ABB RobotStudio station: AssemblyCell_ZZRobotics_final.rspag

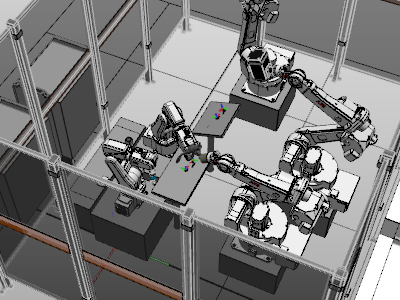
--- station ---
Station Project1 (saved by RobotStudio 22.3.10190.2)
Controller Controller4, task T_ROB2: task frame (RAPID world) sits at (-1070, 1330, 300) mm, rotated rx 0 ry 0 rz -90 deg in the station
Controller Controller4, task T_ROB1: task frame (RAPID world) sits at (-1070, 1330, 300) mm, rotated rx 0 ry 0 rz -90 deg in the station
Controller Controller3, task T_ROB1: task frame (RAPID world) sits at (-374.93, 1144.99, 305) mm, rotated rx 0 ry 0 rz -90 deg in the station
Controller Controller1, task T_ROB2: task frame (RAPID world) sits at (-250, 60, 415.69) mm, rotated rx 0 ry 0 rz 180 deg in the station
Controller Controller1, task T_ROB1: task frame (RAPID world) sits at (-250, 60, 415.69) mm, rotated rx 0 ry 0 rz 180 deg in the station
Controller Controller1
  mechanical unit ROB_1: IRB120_3_58__01_ActLoader, 6 joints, base frame (0, 0, 0) mm
  mechanical unit ROB_2: IRB120_3_58__01_ActTransmitter, 6 joints, base frame (588.39, -10, 0) mm, rotated rx 0 ry 0 rz -90 deg
Controller Controller3
  mechanical unit ROB_1: IRB1520ID_4_150__02_ActWelding, 6 joints, base frame (0, 0, 0) mm
Controller Controller4
  mechanical unit ROB_1: IRB1520ID_4_150__ActDrilling, 6 joints, base frame (0, 0, 0) mm
  mechanical unit ROB_2: IRB1520ID_4_150__ActEndeep, 6 joints, base frame (790, -930, 0) mm, rotated rx 0 ry 0 rz 90 deg
Layout (positions relative to the parent item):
  - RobotBase_Welding [part] at (-620, 914, 10) mm, size 500 x 500 x 300 mm
  - IRB120_3_58__01_ActTransmitter [mechanism, from Robots\IRB120_3_58_G_01.rslib] at (-838.39, 70, 415.69) mm, rotated rx 0 ry 0 rz 90 deg; joint values [-0.5895, 0.4014, 0.0311, 0, 1.1382, -2.1603] (rad or m)
  - IRB120_3_58__01_ActLoader [mechanism, from Robots\IRB120_3_58_G_01.rslib] at (-250, 60, 415.69) mm, rotated rx 0 ry 0 rz 180 deg; joint values [-1.4842, -0.4691, 0.5158, -0.0707, 1.4263, -0.6336] (rad or m)
  - Gripper_Vacuum [mechanism, from Components\smc_gripper.rslib] at (-261.42, 249.64, 930.86) mm, rotated rx -173.43 ry 2.1 rz -48.23 deg
  - Gripper_Fingers [mechanism, from Tools\ABB_Smart_Gripper_Servo_Fingers.rslib] at (-611, 410, 819.18) mm, rotated rx -180 ry 0 rz 0 deg; joint values [0] (rad or m)
  - RA_MTG4000_22 [mechanism, from Tools\Fronius_Robacta_MTG4000_22deg.rslib] at (-374.93, 698.3, 1167.59) mm, rotated rx 180 ry 55 rz 90 deg
  - Table_Welding [graphiccomponentgroup, from Components\Table_Welding.rslib] at (-730, 250, 0) mm
    - TableLeg [part, from Components\Table_Welding.rslib] at (110, 0, 0) mm
    - TablePlate [part, from Components\Table_Welding.rslib] at (730, -250, 0) mm
    - Cylinder_GripWelding_Support [mechanism, from Components\Cylinder.rslib] at (730, -250, 0) mm; joint values [0] (rad or m)
    - Cylinder_GripWelding_Tail [mechanism, from Components\Cylinder.rslib] at (-449, 580, 0) mm, rotated rx 0 ry 0 rz 180 deg; joint values [0] (rad or m)
  - Group_Inlet [graphiccomponentgroup] at (0, 3, 0) mm
    - Desk_L1_H1 [part] at (-279.56, -346.1, 404.98) mm, rotated rx 0 ry 0 rz 90 deg, size 60 x 90 x 5 mm
    - Desk_L2_H2 [part], size 100 x 60 x 5 mm
    - Profile_H1 [part] at (-683.6, -256.15, 395.47) mm, size 45 x 45 x 60 mm
    - Profile_H2 [part], size 45 x 45 x 70 mm
    - Table_Inlet [part] at (0, 40, 0) mm, size 1000 x 257.3 x 400 mm
    - l2_h2_welded [part] at (-595, 407, 640) mm, rotated rx 90 ry 0 rz 90 deg, size 60 x 75 x 100 mm
    - l1_h1_welded [part] at (-590, 407, 640) mm, rotated rx 0 ry 0 rz 90 deg, size 60 x 90 x 65 mm
    - l1_h1_welded_countersink [part] at (-1230, 404.46, 634.13) mm, rotated rx 90 ry -20 rz 90 deg, size 60 x 65 x 90 mm
    - l2_h2_welded_countersink [part] at (-1225, 404.46, 634.13) mm, rotated rx 90 ry -20 rz 90 deg, size 60 x 75 x 100 mm
    - l2_h2_welded_holes [part] at (-1225, 404.46, 634.13) mm, rotated rx 90 ry -20 rz 90 deg, size 60 x 75 x 100 mm
    - l1_h1_welded_holes [part] at (-1230, 404.46, 634.13) mm, rotated rx 90 ry -20 rz 90 deg, size 60 x 65 x 90 mm
    - Desk_L2_H2_1 [part], size 100 x 60 x 5 mm
    - Profile_H2_2 [part], size 45 x 45 x 70 mm
    - Desk_L2_H2_3 [part], size 100 x 60 x 5 mm
    - Profile_H2_4 [part], size 45 x 45 x 70 mm
    - Desk_L2_H2_5 [part], size 100 x 60 x 5 mm
    - Profile_H2_6 [part], size 45 x 45 x 70 mm
  - RobotBase_Transmission [part], size 500 x 500 x 404 mm
  - RobotBase_Loader [part] at (570, 0, 0) mm, size 500 x 500 x 404 mm
  - IRB1520ID_4_150__02_ActWelding [mechanism, from Robots\IRB1520ID_4_150_G_02.rslib] at (-374.93, 1144.99, 305) mm, rotated rx 0 ry 0 rz -90 deg; joint values [0, -1.2217, 1.0472, 0, 0.7854, 0] (rad or m)
  - SmartComponent_ActLoader [smart component]
      signals: DI do_grip_on, DI do_grip_off, DI do_vacuum_on, DI do_vacuum_off
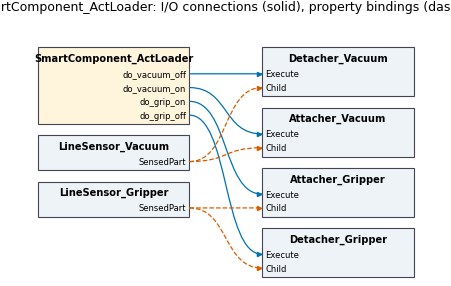
      connections:
        SmartComponent_ActLoader.do_vacuum_off -> Detacher_Vacuum.Execute
        SmartComponent_ActLoader.do_vacuum_on -> Attacher_Vacuum.Execute
        SmartComponent_ActLoader.do_grip_on -> Attacher_Gripper.Execute
        SmartComponent_ActLoader.do_grip_off -> Detacher_Gripper.Execute
        LineSensor_Vacuum.SensedPart => Detacher_Vacuum.Child
        LineSensor_Vacuum.SensedPart => Attacher_Vacuum.Child
        LineSensor_Gripper.SensedPart => Attacher_Gripper.Child
        LineSensor_Gripper.SensedPart => Detacher_Gripper.Child
    - LineSensor_Gripper [smart component, from Components\LineSensor.rslib] at (-611, 410, 704.98) mm, rotated rx -180 ry 0 rz 0 deg
        properties: Start=[0.000368147116492024 0.000112762068043337 -0.00954004890841353]; End=[0.000704727202270661 0.000672266486728079 0.0254538601137482]; Radius=0.005; SensedPart=(none); SensedPoint=[0 0 0]
      - _sensorPart_ [part], size 10.3 x 10.6 x 35.2 mm
    - LineSensor_Vacuum [smart component, from Components\LineSensor.rslib] at (-249.37, 270, 735.28) mm, rotated rx -173.43 ry 2.1 rz -48.23 deg
        properties: Start=[0.000258350395641593 -0.000244336751510213 0.000305598823163056]; End=[0.000624252122424396 0.000899619015264114 0.0102332108789397]; Radius=0.005; SensedPart=(none); SensedPoint=[-0.273905639648438 -0.353316131591797 0.454631866455078]
      - _sensorPart_ [part], size 10.1 x 10.9 x 11.1 mm
    - Attacher_Gripper [smart component, from Components\Attacher.rslib]
        properties: Parent=Gripper_Fingers; Flange=0; Child=(none); Mount=false; Offset=[0 0 0]; Orientation=[0 0 0]
    - Attacher_Vacuum [smart component, from Components\Attacher.rslib]
        properties: Parent=Gripper_Vacuum; Flange=0; Child=(none); Mount=false; Offset=[0 0 0]; Orientation=[0 0 0]
    - Detacher_Gripper [smart component, from Components\Detacher.rslib]
        properties: Child=(none); KeepPosition=true
    - Detacher_Vacuum [smart component, from Components\Detacher.rslib]
        properties: Child=(none); KeepPosition=true
  - SmartComponent_PartsIO [smart component]
      signals: DI spawn_desk_l1_h1, DI spawn_desk_l2_h2, DI spawn_profile_l1_h1, DI spawn_profile_l2_h2, DI spawn_welded_l1_h1, DI spawn_welded_l2_h2, DI spawn_holed_l1_h1, DI spawn_holed_l2_h2, DI drain_desk_l1_h1, DI drain_desk_l2_h2, DI drain_profile_l1_h1, DI drain_profile_l2_h2, DI drain_welded_l1_h1, DI drain_welded_l2_h2, DI drain_holed_l1_h1, DI drain_holed_l2_h2, DI drain_endeep_l2_h2, DI drain_endeep_l1_h1, DI spawn_endeep_l1_h1, DI spawn_endeep_l2_h2
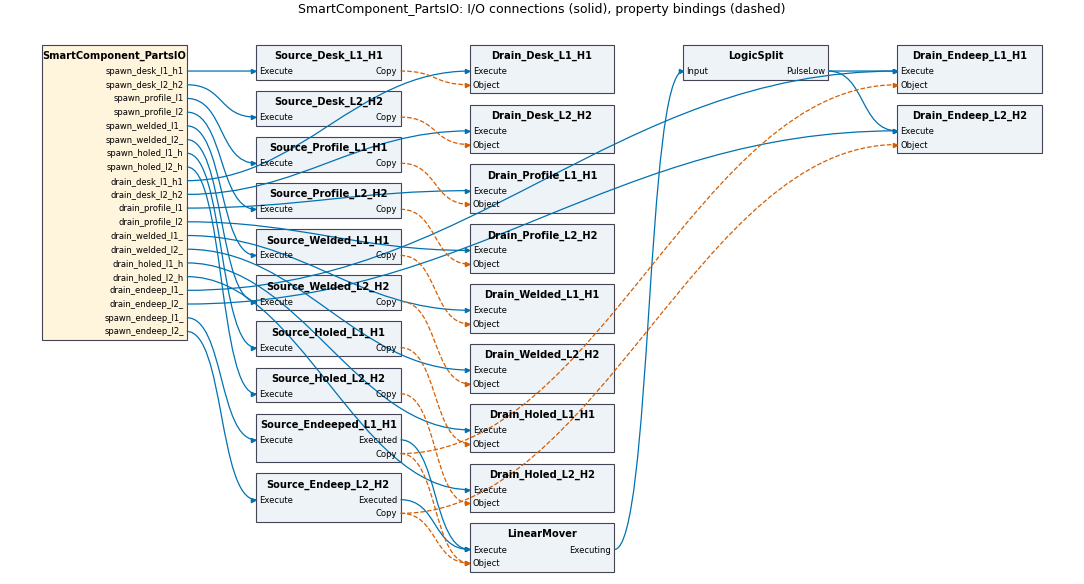
      connections:
        SmartComponent_PartsIO.spawn_desk_l1_h1 -> Source_Desk_L1_H1.Execute
        SmartComponent_PartsIO.spawn_desk_l2_h2 -> Source_Desk_L2_H2.Execute
        SmartComponent_PartsIO.spawn_profile_l1_h1 -> Source_Profile_L1_H1.Execute
        SmartComponent_PartsIO.spawn_profile_l2_h2 -> Source_Profile_L2_H2.Execute
        SmartComponent_PartsIO.spawn_welded_l1_h1 -> Source_Welded_L1_H1.Execute
        SmartComponent_PartsIO.spawn_welded_l2_h2 -> Source_Welded_L2_H2.Execute
        SmartComponent_PartsIO.spawn_holed_l1_h1 -> Source_Holed_L1_H1.Execute
        SmartComponent_PartsIO.spawn_holed_l2_h2 -> Source_Holed_L2_H2.Execute
        SmartComponent_PartsIO.drain_desk_l1_h1 -> Drain_Desk_L1_H1.Execute
        SmartComponent_PartsIO.drain_desk_l2_h2 -> Drain_Desk_L2_H2.Execute
        SmartComponent_PartsIO.drain_profile_l1_h1 -> Drain_Profile_L1_H1.Execute
        SmartComponent_PartsIO.drain_profile_l2_h2 -> Drain_Profile_L2_H2.Execute
        SmartComponent_PartsIO.drain_welded_l1_h1 -> Drain_Welded_L1_H1.Execute
        SmartComponent_PartsIO.drain_welded_l2_h2 -> Drain_Welded_L2_H2.Execute
        SmartComponent_PartsIO.drain_holed_l1_h1 -> Drain_Holed_L1_H1.Execute
        SmartComponent_PartsIO.drain_holed_l2_h2 -> Drain_Holed_L2_H2.Execute
        SmartComponent_PartsIO.drain_endeep_l1_h1 -> Drain_Endeep_L1_H1.Execute
        SmartComponent_PartsIO.drain_endeep_l2_h2 -> Drain_Endeep_L2_H2.Execute
        SmartComponent_PartsIO.spawn_endeep_l1_h1 -> Source_Endeeped_L1_H1.Execute
        SmartComponent_PartsIO.spawn_endeep_l2_h2 -> Source_Endeep_L2_H2.Execute
        Source_Endeep_L2_H2.Executed -> LinearMover.Execute
        Source_Endeeped_L1_H1.Executed -> LinearMover.Execute
        LinearMover.Executing -> LogicSplit.Input
        LogicSplit.PulseLow -> Drain_Endeep_L1_H1.Execute
        LogicSplit.PulseLow -> Drain_Endeep_L2_H2.Execute
        Source_Desk_L1_H1.Copy => Drain_Desk_L1_H1.Object
        Source_Desk_L2_H2.Copy => Drain_Desk_L2_H2.Object
        Source_Profile_L1_H1.Copy => Drain_Profile_L1_H1.Object
        Source_Profile_L2_H2.Copy => Drain_Profile_L2_H2.Object
        Source_Welded_L1_H1.Copy => Drain_Welded_L1_H1.Object
        Source_Welded_L2_H2.Copy => Drain_Welded_L2_H2.Object
        Source_Holed_L1_H1.Copy => Drain_Holed_L1_H1.Object
        Source_Holed_L2_H2.Copy => Drain_Holed_L2_H2.Object
        Source_Endeeped_L1_H1.Copy => Drain_Endeep_L1_H1.Object
        Source_Endeep_L2_H2.Copy => Drain_Endeep_L2_H2.Object
        Source_Endeeped_L1_H1.Copy => LinearMover.Object
        Source_Endeep_L2_H2.Copy => LinearMover.Object
    - Source_Desk_L1_H1 [smart component, from Components\Source.rslib] at (-294.16, -347, 399.98) mm, rotated rx 0 ry 0 rz 90 deg
        properties: Source=Desk_L1_H1; Copy=(none); Parent=(none); Position=[-0.279564 -0.346 0.404979]; Orientation=[0 0 1.5707963267949]; Transient=true; PhysicsBehavior=-1
    - Source_Desk_L2_H2 [smart component, from Components\Source.rslib]
        properties: Source=Desk_L2_H2; Copy=(none); Parent=(none); Position=[0 0 0]; Orientation=[0 0 0]; Transient=true; PhysicsBehavior=-1
    - Source_Profile_L1_H1 [smart component, from Components\Source.rslib]
        properties: Source=Profile_H1; Copy=(none); Parent=(none); Position=[-0.683597 -0.256153 0.395473]; Orientation=[0 0 0]; Transient=true; PhysicsBehavior=-1
    - Source_Profile_L2_H2 [smart component, from Components\Source.rslib]
        properties: Source=Profile_H2; Copy=(none); Parent=(none); Position=[0 0 0]; Orientation=[0 0 0]; Transient=true; PhysicsBehavior=-1
    - Source_Welded_L1_H1 [smart component, from Components\Source.rslib]
        properties: Source=l1_h1_welded; Copy=(none); Parent=(none); Position=[-0.59 0.407 0.64]; Orientation=[0 0 1.5707963267949]; Transient=true; PhysicsBehavior=-1
    - Source_Welded_L2_H2 [smart component, from Components\Source.rslib]
        properties: Source=l2_h2_welded; Copy=(none); Parent=(none); Position=[-0.595 0.407 0.64]; Orientation=[1.5707963267949 0 1.5707963267949]; Transient=true; PhysicsBehavior=-1
    - Source_Holed_L1_H1 [smart component, from Components\Source.rslib]
        properties: Source=l1_h1_welded_holes; Copy=(none); Parent=(none); Position=[-1.23 0.404459 0.634127]; Orientation=[1.5707963267949 -0.349065850398866 1.5707963267949]; Transient=true; PhysicsBehavior=-1
    - Source_Holed_L2_H2 [smart component, from Components\Source.rslib]
        properties: Source=l2_h2_welded_holes; Copy=(none); Parent=(none); Position=[-1.225 0.404459 0.634127]; Orientation=[1.5707963267949 -0.349065850398866 1.5707963267949]; Transient=true; PhysicsBehavior=-1
    - Drain_Desk_L1_H1 [smart component, from Components\Sink.rslib]
        properties: Object=(none)
    - Drain_Holed_L1_H1 [smart component, from Components\Sink.rslib]
        properties: Object=(none)
    - Drain_Profile_L2_H2 [smart component, from Components\Sink.rslib]
        properties: Object=(none)
    - Drain_Profile_L1_H1 [smart component, from Components\Sink.rslib]
        properties: Object=(none)
    - Drain_Welded_L2_H2 [smart component, from Components\Sink.rslib]
        properties: Object=(none)
    - Drain_Desk_L2_H2 [smart component, from Components\Sink.rslib]
        properties: Object=(none)
    - Drain_Holed_L2_H2 [smart component, from Components\Sink.rslib]
        properties: Object=(none)
    - Drain_Welded_L1_H1 [smart component, from Components\Sink.rslib]
        properties: Object=(none)
    - Source_Endeeped_L1_H1 [smart component, from Components\Source.rslib]
        properties: Source=l1_h1_welded_countersink; Copy=(none); Parent=(none); Position=[-1.23 0.404459 0.634127]; Orientation=[1.5707963267949 -0.349065850398866 1.5707963267949]; Transient=true; PhysicsBehavior=-1
    - Source_Endeep_L2_H2 [smart component, from Components\Source.rslib]
        properties: Source=l2_h2_welded_countersink; Copy=(none); Parent=(none); Position=[-1.225 0.404459 0.634127]; Orientation=[1.5707963267949 -0.349065850398866 1.5707963267949]; Transient=true; PhysicsBehavior=-1
    - Drain_Endeep_L2_H2 [smart component, from Components\Sink.rslib]
        properties: Object=(none)
    - Drain_Endeep_L1_H1 [smart component, from Components\Sink.rslib]
        properties: Object=(none)
    - LinearMover [smart component, from Components\LinearMover2.rslib]
        properties: Object=(none); Direction=[-0.1 0 0]; Distance=0.17; Duration=2; Reference=Local; ReferenceObject=(none)
    - LogicSplit [smart component, from Components\LogicSplit.rslib]
  - LogicGate [smart component, from Components\LogicGate.rslib]
      properties: Operator=AND; Delay=0
  - LogicGate_2 [smart component, from Components\LogicGate.rslib]
      properties: Operator=AND; Delay=0
  - LogicGate_3 [smart component, from Components\LogicGate.rslib]
      properties: Operator=AND; Delay=0
  - LogicGate_4 [smart component, from Components\LogicGate.rslib]
      properties: Operator=AND; Delay=0
  - Group_Drill_Endeep_Cell [graphiccomponentgroup]
    - RobotBase_Endeep [part] at (-1760, 283.99, 10) mm, rotated rx 0 ry 0 rz 90 deg, size 500 x 500 x 300 mm
    - RobotBase_Drilling [part] at (-1320, 1114, 10) mm, size 500 x 500 x 300 mm
    - Table_Drilling [graphiccomponentgroup] at (-1370, 250, 0) mm, rotated rx 20 ry 0 rz 0 deg
      - TableLeg [part] at (60, 0, 0) mm, rotated rx -20 ry 0 rz 0 deg, size 60 x 60 x 600 mm
      - TablePlate [part, from Components\TablePlate.rslib] at (1240, -234.92, 85.51) mm, rotated rx -20 ry 0 rz 0 deg
    - Cylinder_GripDrilling_Support [mechanism, from Components\Cylinder_1.rslib] at (-640, 240.97, -107.21) mm, rotated rx 20 ry 0 rz 0 deg; joint values [0] (rad or m)
    - Cylinder_GripDrilling_Tail [mechanism, from Components\Cylinder_1.rslib] at (-1819.91, 1021, 176.44) mm, rotated rx -20 ry 0 rz 180 deg; joint values [0] (rad or m)
    - Drill_Tool [mechanism, from Components\Drill_Tool.rslib] at (-1079.95, 911.09, 1539.96) mm, rotated rx -180 ry -70 rz -90 deg
    - Endeep_Tool [mechanism, from Components\Endeep_Tool.rslib] at (-1432.49, 333.31, 1851.39) mm, rotated rx 0 ry -70 rz -90 deg
  - IRB1520ID_4_150__ActDrilling [mechanism, from Robots\IRB1520ID_4_150_G_02.rslib] at (-1070, 1330, 300) mm, rotated rx 0 ry 0 rz -90 deg; joint values [-0.0458, -0.9578, 0.4598, 0.0574, 0.8482, -0.0537] (rad or m)
  - IRB1520ID_4_150__ActEndeep [mechanism, from Robots\IRB1520ID_4_150_G_02.rslib] at (-2000, 540, 300) mm; joint values [-0.6243, -0.1174, -0.2377, 2.1619, 1.978, -0.9764] (rad or m)
  - LogicGate_5 [smart component, from Components\LogicGate.rslib]
      properties: Operator=AND; Delay=0
  - LogicGate_6 [smart component, from Components\LogicGate.rslib]
      properties: Operator=AND; Delay=0
  - LogicGate_7 [smart component, from Components\LogicGate.rslib]
      properties: Operator=AND; Delay=0
  - LogicGate_8 [smart component, from Components\LogicGate.rslib]
      properties: Operator=AND; Delay=0
  - SmartComponent_Cylinders [smart component]
      signals: DI open_weld_support, DI open_weld_tail, DI open_drill_support, DI open_drill_tail, DI close_weld_support, DI close_weld_tail, DI close_drill_support, DI close_drill_tail
      connections:
        SmartComponent_Cylinders.open_drill_support -> PoseMover.Execute
        SmartComponent_Cylinders.close_drill_support -> PoseMover_2.Execute
        SmartComponent_Cylinders.open_drill_tail -> PoseMover_7.Execute
        SmartComponent_Cylinders.close_drill_tail -> PoseMover_3.Execute
        SmartComponent_Cylinders.open_weld_support -> PoseMover_6.Execute
        SmartComponent_Cylinders.close_weld_support -> PoseMover_4.Execute
        SmartComponent_Cylinders.open_weld_tail -> PoseMover_5.Execute
        SmartComponent_Cylinders.close_weld_tail -> PoseMover_8.Execute
    - PoseMover [smart component, from Components\PoseMover.rslib]
        properties: Mechanism=Cylinder_GripDrilling_Support; Pose=1; Duration=0
    - PoseMover_2 [smart component, from Components\PoseMover.rslib]
        properties: Mechanism=Cylinder_GripDrilling_Support; Pose=2; Duration=0
    - PoseMover_3 [smart component, from Components\PoseMover.rslib]
        properties: Mechanism=Cylinder_GripDrilling_Tail; Pose=2; Duration=0
    - PoseMover_4 [smart component, from Components\PoseMover.rslib]
        properties: Mechanism=Cylinder_GripWelding_Support; Pose=2; Duration=0
    - PoseMover_5 [smart component, from Components\PoseMover.rslib]
        properties: Mechanism=Cylinder_GripWelding_Tail; Pose=1; Duration=0
    - PoseMover_6 [smart component, from Components\PoseMover.rslib]
        properties: Mechanism=Cylinder_GripWelding_Support; Pose=1; Duration=0
    - PoseMover_7 [smart component, from Components\PoseMover.rslib]
        properties: Mechanism=Cylinder_GripDrilling_Tail; Pose=1; Duration=0
    - PoseMover_8 [smart component, from Components\PoseMover.rslib]
        properties: Mechanism=Cylinder_GripWelding_Tail; Pose=2; Duration=0
  - Fence [graphiccomponentgroup] at (0, 201.34, 0) mm
    - Z_Fence_800 [part] at (-2692.2, -847.39, 0) mm, size 159.8 x 979.2 x 2218.8 mm
    - Z_Fence_802 [part] at (-2692.2, 12.61, 0) mm, size 159.8 x 979.2 x 2218.8 mm
    - Z_Fence_806 [part] at (-2692.2, 872.87, 0) mm, size 159.8 x 979.2 x 2218.8 mm
    - Z_Fence_808 [part] at (-974.44, -853.03, 0) mm, rotated rx 0 ry 0 rz 90 deg, size 159.8 x 979.2 x 2218.8 mm
    - Z_Fence_809 [part] at (-1834.6, -853.03, 0) mm, rotated rx 0 ry 0 rz 90 deg, size 159.8 x 979.2 x 2218.8 mm
    - Z_Fence_810 [part] at (-114.19, -853.03, 0) mm, rotated rx 0 ry 0 rz 90 deg, size 159.8 x 979.2 x 2218.8 mm
    - Z_Fence_811 [part] at (745.69, -853.03, 0) mm, rotated rx 0 ry 0 rz 90 deg, size 159.8 x 979.2 x 2218.8 mm
    - Z_Fence_813 [part] at (-2691.02, 1743.1, 0) mm, rotated rx 0 ry 0 rz -90 deg, size 159.8 x 979.2 x 2218.8 mm
    - Z_Fence_814 [part] at (-1830.85, 1743.1, 0) mm, rotated rx 0 ry 0 rz -90 deg, size 159.8 x 979.2 x 2218.8 mm
    - Z_Fence_815 [part] at (-110.06, 1743.1, 0) mm, rotated rx 0 ry 0 rz -90 deg, size 159.8 x 979.2 x 2218.8 mm
    - Z_Fence_816 [part] at (-970.7, 1743.1, 0) mm, rotated rx 0 ry 0 rz -90 deg, size 159.8 x 979.2 x 2218.8 mm
    - Z_Fence_818 [part] at (749.49, 1737.83, 0) mm, rotated rx 0 ry 0 rz 180 deg, size 159.8 x 979.2 x 2218.8 mm
    - Z_Fence_819 [part] at (749.49, 877.62, 0) mm, rotated rx 0 ry 0 rz 180 deg, size 159.8 x 979.2 x 2218.8 mm
    - Z_Fence_820 [part] at (749.49, 17.63, 0) mm, rotated rx 0 ry 0 rz 180 deg, size 159.8 x 979.2 x 2218.8 mm
  - _Skrine [graphiccomponentgroup]
    - OmniCore V250XT [mechanism, from %ABB.RobotStudio.Models.OmniCore%\OmniCore_V250XT.rslib] at (-135.27, 2273.01, 0) mm, rotated rx 0 ry 0 rz 180 deg; joint values [0] (rad or m)
    - OmniCore V250XT_2 [mechanism, from %ABB.RobotStudio.Models.OmniCore%\OmniCore_V250XT.rslib] at (-930.19, 2273.01, 0) mm, rotated rx 0 ry 0 rz 180 deg; joint values [0] (rad or m)
    - OmniCore V250XT_3 [mechanism, from %ABB.RobotStudio.Models.OmniCore%\OmniCore_V250XT.rslib] at (-1769.47, 2273.01, 0) mm, rotated rx 0 ry 0 rz 180 deg; joint values [0] (rad or m)
    - OmniCore V250XT_4 [mechanism, from %ABB.RobotStudio.Models.OmniCore%\OmniCore_V250XT.rslib] at (-51.9, -1005.58, 0) mm; joint values [0] (rad or m)
    - OmniCore V250XT_5 [mechanism, from %ABB.RobotStudio.Models.OmniCore%\OmniCore_V250XT.rslib] at (-880.12, -1005.58, 0) mm; joint values [0] (rad or m)
Attachment: Gripper_Vacuum is attached to IRB120_3_58__01_ActLoader / Link6
Attachment: Gripper_Fingers is attached to IRB120_3_58__01_ActTransmitter / Link6
Attachment: RA_MTG4000_22 is attached to IRB1520ID_4_150__02_ActWelding / Link6
Attachment: LineSensor_Gripper is attached to Gripper_Fingers / HandBase
Attachment: LineSensor_Vacuum is attached to Gripper_Vacuum / Assembly_ABBGRIP_2
Attachment: Drill_Tool is attached to IRB1520ID_4_150__ActDrilling / Link6
Attachment: Endeep_Tool is attached to IRB1520ID_4_150__ActEndeep / Link6
Station signals: DI p_type_1_small, DI p_type_2_big, DI produce
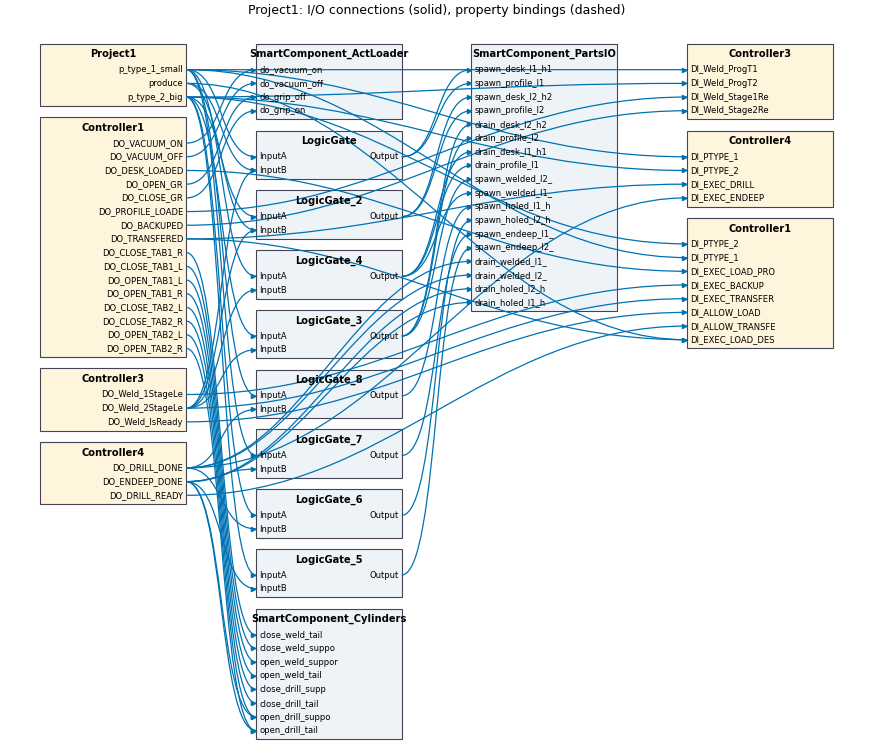
Station logic (signal -> signal, property => property):
  Project1.p_type_1_small -> LogicGate.InputA
  Project1.produce -> LogicGate.InputB
  LogicGate.Output -> SmartComponent_PartsIO.spawn_desk_l1_h1
  LogicGate.Output -> SmartComponent_PartsIO.spawn_profile_l1_h1
  Project1.p_type_2_big -> LogicGate_2.InputA
  Project1.produce -> LogicGate_2.InputB
  LogicGate_2.Output -> SmartComponent_PartsIO.spawn_desk_l2_h2
  LogicGate_2.Output -> SmartComponent_PartsIO.spawn_profile_l2_h2
  Controller1.DO_VACUUM_ON -> SmartComponent_ActLoader.do_vacuum_on
  Controller1.DO_VACUUM_OFF -> SmartComponent_ActLoader.do_vacuum_off
  Project1.p_type_2_big -> Controller1.DI_PTYPE_2
  Project1.p_type_1_small -> Controller1.DI_PTYPE_1
  Controller1.DO_DESK_LOADED -> Controller1.DI_EXEC_LOAD_PROFILE
  Controller1.DO_OPEN_GR -> SmartComponent_ActLoader.do_grip_off
  Controller1.DO_CLOSE_GR -> SmartComponent_ActLoader.do_grip_on
  Project1.p_type_1_small -> Controller3.DI_Weld_ProgT1
  Project1.p_type_2_big -> Controller3.DI_Weld_ProgT2
  Controller1.DO_PROFILE_LOADED -> Controller3.DI_Weld_Stage1Req
  Controller3.DO_Weld_1StageLeave -> Controller1.DI_EXEC_BACKUP
  Controller1.DO_BACKUPED -> Controller3.DI_Weld_Stage2Req
  Controller3.DO_Weld_2StageLeave -> Controller1.DI_EXEC_TRANSFER
  Project1.p_type_2_big -> LogicGate_3.InputA
  Controller3.DO_Weld_2StageLeave -> LogicGate_3.InputB
  LogicGate_3.Output -> SmartComponent_PartsIO.drain_desk_l2_h2
  LogicGate_3.Output -> SmartComponent_PartsIO.drain_profile_l2_h2
  Project1.p_type_1_small -> LogicGate_4.InputA
  Controller3.DO_Weld_2StageLeave -> LogicGate_4.InputB
  LogicGate_4.Output -> SmartComponent_PartsIO.drain_desk_l1_h1
  LogicGate_4.Output -> SmartComponent_PartsIO.drain_profile_l1_h1
  LogicGate_3.Output -> SmartComponent_PartsIO.spawn_welded_l2_h2
  LogicGate_4.Output -> SmartComponent_PartsIO.spawn_welded_l1_h1
  Project1.p_type_1_small -> Controller4.DI_PTYPE_1
  Project1.p_type_2_big -> Controller4.DI_PTYPE_2
  Controller1.DO_TRANSFERED -> Controller4.DI_EXEC_DRILL
  Controller4.DO_DRILL_DONE -> Controller4.DI_EXEC_ENDEEP
  Project1.p_type_1_small -> LogicGate_8.InputA
  Project1.p_type_2_big -> LogicGate_6.InputA
  Controller4.DO_DRILL_DONE -> LogicGate_8.InputB
  Controller4.DO_DRILL_DONE -> LogicGate_6.InputB
  Project1.p_type_1_small -> LogicGate_7.InputA
  Project1.p_type_2_big -> LogicGate_5.InputA
  Controller4.DO_ENDEEP_DONE -> LogicGate_7.InputB
  Controller4.DO_ENDEEP_DONE -> LogicGate_5.InputB
  LogicGate_8.Output -> SmartComponent_PartsIO.spawn_holed_l1_h1
  LogicGate_6.Output -> SmartComponent_PartsIO.spawn_holed_l2_h2
  LogicGate_7.Output -> SmartComponent_PartsIO.spawn_endeep_l1_h1
  LogicGate_5.Output -> SmartComponent_PartsIO.spawn_endeep_l2_h2
  Controller1.DO_CLOSE_TAB1_R -> SmartComponent_Cylinders.close_weld_tail
  Controller1.DO_CLOSE_TAB1_L -> SmartComponent_Cylinders.close_weld_support
  Controller1.DO_OPEN_TAB1_L -> SmartComponent_Cylinders.open_weld_support
  Controller1.DO_OPEN_TAB1_R -> SmartComponent_Cylinders.open_weld_tail
  Controller1.DO_CLOSE_TAB2_L -> SmartComponent_Cylinders.close_drill_support
  Controller1.DO_CLOSE_TAB2_R -> SmartComponent_Cylinders.close_drill_tail
  Controller1.DO_OPEN_TAB2_L -> SmartComponent_Cylinders.open_drill_support
  Controller1.DO_OPEN_TAB2_R -> SmartComponent_Cylinders.open_drill_tail
  Controller4.DO_ENDEEP_DONE -> SmartComponent_Cylinders.open_drill_tail
  Controller4.DO_ENDEEP_DONE -> SmartComponent_Cylinders.open_drill_support
  Controller3.DO_Weld_IsReady -> Controller1.DI_ALLOW_LOAD
  Controller3.DO_Weld_2StageLeave -> LogicGate_2.InputB
  Controller3.DO_Weld_2StageLeave -> LogicGate.InputB
  Controller4.DO_DRILL_READY -> Controller1.DI_ALLOW_TRANSFER
  Project1.produce -> Controller1.DI_EXEC_LOAD_DESK
  Controller1.DO_TRANSFERED -> Controller1.DI_EXEC_LOAD_DESK
  Controller4.DO_DRILL_DONE -> SmartComponent_PartsIO.drain_welded_l1_h1
  Controller4.DO_DRILL_DONE -> SmartComponent_PartsIO.drain_welded_l2_h2
  Controller4.DO_ENDEEP_DONE -> SmartComponent_PartsIO.drain_holed_l2_h2
  Controller4.DO_ENDEEP_DONE -> SmartComponent_PartsIO.drain_holed_l1_h1
Targets, tools, work objects and paths stored in the station and not in the controller backup, written as RAPID:
! task T_ROB2
MODULE Module1
  CONST num WaitGripper:=1;
ENDMODULE


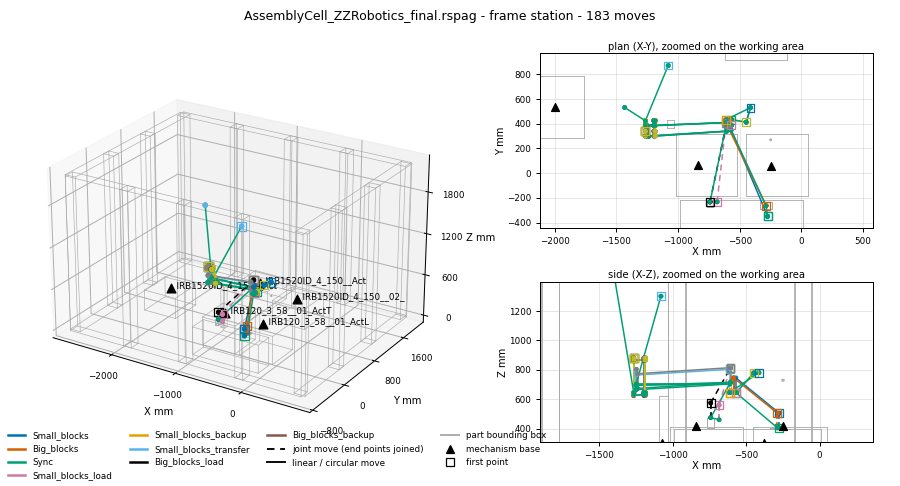
[picture p0: tool path of AssemblyCell_ZZRobotics_final.rspag in frame station, 183 of 212 moves have a stored position in this frame; points joined in program order, loops and branches not executed]
--- Controller Data/Controller1/RAPID/TASK1/PROGMOD/CalibData.mod ---
MODULE CalibData
    PERS tooldata Gripper_Vacuum:=[TRUE,[[0,0.004,197.001],[1,0,0,0]],[1,[0.207,-0.496,71.18],[1,0,0,0],0,0,0]];
ENDMODULE

--- Controller Data/Controller1/RAPID/TASK1/PROGMOD/Module1.mod ---
MODULE Module1
    CONST jointtarget Target_JHome:=[[-85.037200714,-26.876673148,29.555461388,-4.048831126,81.721717608,-36.301936344],[9E+09,9E+09,9E+09,9E+09,9E+09,9E+09]];

    CONST robtarget Target_Base_l2_h2:=[[36.607,323.865,-10.716],[0,0,1,0],[0,0,0,0],[9E+09,9E+09,9E+09,9E+09,9E+09,9E+09]];
    CONST robtarget Target_Base_l1_h1:=[[24.164,410,-10.605],[0,0,1,0],[0,0,1,0],[9E+09,9E+09,9E+09,9E+09,9E+09,9E+09]];

    CONST robtarget Target_Table1_l2_h2_pre:=[[335,-293,229.805],[0,0,1,0],[-1,-1,0,0],[9E+09,9E+09,9E+09,9E+09,9E+09,9E+09]];
    CONST robtarget Target_Table1_l2_h2:=[[335,-346.85,229.340933033],[0,0,1,0],[-1,-1,0,0],[9E+09,9E+09,9E+09,9E+09,9E+09,9E+09]];

    CONST robtarget Target_Table1_l1_h1_pre:=[[319.886,-290.252,229.772],[0,0,1,0],[0,0,0,0],[9E+09,9E+09,9E+09,9E+09,9E+09,9E+09]];
    CONST robtarget Target_Table1_l1_h1:=[[334.586,-342.952,229.372],[0,0,1,0],[0,0,0,0],[9E+09,9E+09,9E+09,9E+09,9E+09,9E+09]];

    VAR bool cold_start:=TRUE;
    CONST num wait_vacuum:=1;

    PROC main()
        IF cold_start THEN
            Init;
            cold_start:=FALSE;
        ENDIF

        WaitDI DI_EXEC_LOAD_DESK,1;
        WaitDI DI_ALLOW_LOAD,1;

        IF TestDI(DI_PTYPE_1) THEN
            Small_blocks;
        ELSEIF TestDI(DI_PTYPE_2) THEN
            Big_blocks;
        ELSE
            RETURN ;
        ENDIF
    ENDPROC

    PROC Init()
        PulseDO DO_OPEN_TAB1_L;
        PulseDO DO_OPEN_TAB1_R;
        MoveAbsJ Target_JHome,v1000,fine,Gripper_Vacuum\WObj:=wobj0;
    ENDPROC

    PROC Small_blocks()
        MoveJ Offs(Target_Base_l1_h1,0,0,100),v1000,fine,Gripper_Vacuum;
        MoveJ Offs(Target_Base_l1_h1,0,0,0),v1000,fine,Gripper_Vacuum;

        !Attach %%%%%%%%%%%%%%%%%%%%%%%%%%%%%%%%%%%%%%
        PulseDO DO_VACUUM_ON;
        WaitTime wait_vacuum;

        MoveJ Offs(Target_Base_l1_h1,0,0,100),v1000,fine,Gripper_Vacuum;
        MoveL Offs(Target_Table1_l1_h1_pre,0,0,100),v1000,fine,Gripper_Vacuum;
        WaitTime 0.5;
        MoveL Offs(Target_Table1_l1_h1_pre,0,0,0),v200,fine,Gripper_Vacuum;
        WaitTime 0.5;
        MoveL Offs(Target_Table1_l1_h1,0,0,0),v200,fine,Gripper_Vacuum;

        WaitTime 0.5;
        PulseDO DO_CLOSE_TAB1_L;
        PulseDO DO_CLOSE_TAB1_R;

        !Detach %%%%%%%%%%%%%%%%
        PulseDO DO_VACUUM_OFF;
        WaitTime wait_vacuum;

        MoveL Offs(Target_Table1_l1_h1,0,0,100),v200,fine,Gripper_Vacuum;
        MoveAbsJ Target_JHome,v1000,fine,Gripper_Vacuum\WObj:=wobj0;

        PulseDO DO_DESK_LOADED;
    ENDPROC

    PROC Big_blocks()
        MoveJ Offs(Target_Base_l2_h2,0,0,100),v1000,fine,Gripper_Vacuum;
        MoveJ Offs(Target_Base_l2_h2,0,0,0),v1000,fine,Gripper_Vacuum;

        !Attach %%%%%%%%%%%%%%%%%%%%%%%%%%%%%%%%%%%%%%
        PulseDO DO_VACUUM_ON;
        WaitTime wait_vacuum;

        MoveJ Offs(Target_Base_l2_h2,0,0,100),v1000,fine,Gripper_Vacuum;
        MoveL Offs(Target_Table1_l2_h2_pre,0,0,100),v1000,fine,Gripper_Vacuum;
        WaitTime 0.5;
        MoveL Offs(Target_Table1_l2_h2_pre,0,0,0),v200,fine,Gripper_Vacuum;
        WaitTime 0.5;
        MoveL Offs(Target_Table1_l2_h2,0,0,0),v200,fine,Gripper_Vacuum;

        WaitTime 0.5;
        PulseDO DO_CLOSE_TAB1_L;
        PulseDO DO_CLOSE_TAB1_R;

        !Detach %%%%%%%%%%%%%%%%
        PulseDO DO_VACUUM_OFF;
        WaitTime wait_vacuum;

        MoveL Offs(Target_Table1_l2_h2,0,0,100),v200,fine,Gripper_Vacuum;
        MoveAbsJ Target_JHome,v1000,fine,Gripper_Vacuum\WObj:=wobj0;

        PulseDO DO_DESK_LOADED;
    ENDPROC

    PROC Sync()
        MoveAbsJ Target_JHome,v1000,fine,Gripper_Vacuum\WObj:=wobj0;
        MoveL Target_Base_l1_h1,v1000,z100,Gripper_Vacuum\WObj:=wobj0;
        MoveL Target_Base_l2_h2,v1000,z100,Gripper_Vacuum\WObj:=wobj0;
        MoveL Target_Table1_l1_h1_pre,v1000,z100,Gripper_Vacuum\WObj:=wobj0;
        MoveL Target_Table1_l1_h1,v1000,z100,Gripper_Vacuum\WObj:=wobj0;
        MoveL Target_Table1_l2_h2_pre,v1000,z100,Gripper_Vacuum\WObj:=wobj0;
        MoveL Target_Table1_l2_h2,v1000,z100,Gripper_Vacuum\WObj:=wobj0;
    ENDPROC
ENDMODULE

--- Controller Data/Controller1/RAPID/TASK2/PROGMOD/CalibData.mod ---
MODULE CalibData
    PERS tooldata Gripper_Fingers:=[TRUE,[[0,0,114.2],[1,0,0,0]],[0.215,[8.7,12.3,49.2],[1,0,0,0],0.00021,0.00024,0.00009]];
ENDMODULE

--- Controller Data/Controller1/RAPID/TASK2/PROGMOD/Module1.mod ---
MODULE Module1
    CONST jointtarget Target_JHome:=[[-26.597577745,-44.264017247,35.261659694,-19.248693519,81.614947173,-88.381493558],[9E+09,9E+09,9E+09,9E+09,9E+09,9E+09]];

    CONST robtarget Target_Base_l2_h2:=[[490.966,292.847,59.284],[0,0.707106781,0.707106781,0],[-2,0,0,0],[9E+09,9E+09,9E+09,9E+09,9E+09,9E+09]];
    CONST robtarget Target_Base_l1_h1:=[[433.597,292.153,44.778],[0,0.707106781,0.707106781,0],[-2,0,1,0],[9E+09,9E+09,9E+09,9E+09,9E+09,9E+09]];

    CONST robtarget Target_Table1_l1_h1_takeout:=[[360.972830849,-280.009480233,288.1717752],[0.004810357,-0.000232941,0.999956482,-0.007990003],[-1,0,-2,0],[9E+09,9E+09,9E+09,9E+09,9E+09,9E+09]];
    CONST robtarget Target_Table1_l2_h2_takeout:=[[356,-280,299.305],[0,0,1,0],[-1,0,-2,0],[9E+09,9E+09,9E+09,9E+09,9E+09,9E+09]];

    CONST robtarget Target_Table1_l2_h2:=[[356,-350,299.305],[0,0,1,0],[-1,0,-2,0],[9E+09,9E+09,9E+09,9E+09,9E+09,9E+09]];
    CONST robtarget Target_Table1_l1_h1:=[[361,-350.001,289.29],[0,0,1,0],[-1,0,-2,0],[9E+09,9E+09,9E+09,9E+09,9E+09,9E+09]];

    CONST robtarget Target_Table2_l1_h1:=[[1001,-325.091129765,279.687062196],[0,0,0.984807753,-0.173648178],[0,-1,0,0],[9E+09,9E+09,9E+09,9E+09,9E+09,9E+09]];
    CONST robtarget Target_Table2_l2_h2:=[[996,-321.807256971,288.908661883],[0,0,0.984807753,-0.173648178],[0,0,0,0],[9E+09,9E+09,9E+09,9E+09,9E+09,9E+09]];

    CONST robtarget Target_Table2_l2_h2_takeout:=[[988.5,-237.234921117,258.126848932],[0,0,0.984807753,-0.173648178],[0,0,0,0],[9E+09,9E+09,9E+09,9E+09,9E+09,9E+09]];
    CONST robtarget Target_Table2_l1_h1_takeout:=[[999.5,-240.655323444,248.729567219],[0,0,0.984807753,-0.173648178],[0,-1,0,0],[9E+09,9E+09,9E+09,9E+09,9E+09,9E+09]];

    VAR bool cold_start:=TRUE;
    CONST num wait_gripper:=1;

    PROC main()
        IF cold_start THEN
            Init;
            cold_start:=FALSE;
        ENDIF

        WaitDI DI_EXEC_LOAD_PROFILE,1;
        WaitDI DI_ALLOW_LOAD,1;

        IF TestDI(DI_PTYPE_1) THEN
            Small_blocks_load;
            WaitDI DI_EXEC_BACKUP,1;
            Small_blocks_backup;
            WaitDI DI_EXEC_TRANSFER,1;
            WaitDI DI_ALLOW_TRANSFER,1;
            Small_blocks_transfer;
        ELSEIF TestDI(DI_PTYPE_2) THEN
            Big_blocks_load;
            WaitDI DI_EXEC_BACKUP,1;
            Big_blocks_backup;
            WaitDI DI_EXEC_TRANSFER,1;
            WaitDI DI_ALLOW_TRANSFER,1;
            Big_blocks_transfer;
        ELSE
            RETURN ;
        ENDIF
    ENDPROC

    PROC Init()
        PulseDO DO_OPEN_GR;
        PulseDO DO_OPEN_TAB2_L;
        PulseDO DO_OPEN_TAB2_R;

        MoveAbsJ Target_JHome,v1000,fine,Gripper_Fingers\WObj:=wobj0;
    ENDPROC

    PROC Small_blocks_load()
        MoveJ Offs(Target_Base_l1_h1,0,0,100),v1000,fine,Gripper_Fingers;

        !OPEN Gripper
        PulseDO DO_OPEN_GR;
        WaitTime wait_gripper;

        MoveJ Offs(Target_Base_l1_h1,0,0,0),v1000,fine,Gripper_Fingers;

        !Close gripper
        PulseDO DO_CLOSE_GR;
        WaitTime wait_gripper;

        MoveJ Offs(Target_Base_l1_h1,0,0,100),v1000,fine,Gripper_Fingers;
        MoveJ Offs(Target_Table1_l1_h1,0,0,100),v1000,fine,Gripper_Fingers;
        MoveJ Target_Table1_l1_h1,v200,fine,Gripper_Fingers;
        WaitTime 0.5;

        PulseDO DO_PROFILE_LOADED;
    ENDPROC

    PROC Small_blocks_backup()
        !OPEN Gripper
        PulseDO DO_OPEN_GR;
        WaitTime wait_gripper;

        MoveJ Offs(Target_Table1_l1_h1,0,0,100),v200,fine,Gripper_Fingers;
        MoveAbsJ Target_JHome,v1000,fine,Gripper_Fingers\WObj:=wobj0;

        PulseDO DO_BACKUPED;
    ENDPROC

    PROC Small_blocks_transfer()
        !OPEN Gripper
        PulseDO DO_OPEN_GR;
        WaitTime wait_gripper;

        MoveJ Offs(Target_Table1_l1_h1,0,0,100),v1000,fine,Gripper_Fingers;
        MoveJ Target_Table1_l1_h1,v200,fine,Gripper_Fingers;
        WaitTime 0.5;

        PulseDO DO_OPEN_TAB1_L;
        PulseDO DO_OPEN_TAB1_R;

        !Close gripper
        PulseDO DO_CLOSE_GR;
        WaitTime wait_gripper;

        MoveL Target_Table1_l1_h1_takeout,v200,fine,Gripper_Fingers;
        MoveL Offs(Target_Table1_l1_h1_takeout,0,0,100),v1000,fine,Gripper_Fingers;

        MoveL Offs(Target_Table2_l1_h1_takeout,0,0,100),v1000,fine,Gripper_Fingers;
        MoveL Offs(Target_Table2_l1_h1_takeout,0,0,0),v200,fine,Gripper_Fingers;
        MoveL Offs(Target_Table2_l1_h1,0,0,0),v200,fine,Gripper_Fingers;
        WaitTime 0.5;

        PulseDO DO_CLOSE_TAB2_L;
        PulseDO DO_CLOSE_TAB2_R;

        PulseDO DO_OPEN_GR;
        WaitTime wait_gripper;

        MoveL Offs(Target_Table2_l1_h1,0,0,100),v1000,fine,Gripper_Fingers;
        MoveAbsJ Target_JHome,v1000,fine,Gripper_Fingers\WObj:=wobj0;

        PulseDO DO_TRANSFERED;
    ENDPROC

    PROC Big_blocks_load()
        MoveJ Offs(Target_Base_l2_h2,0,0,100),v1000,fine,Gripper_Fingers;

        !OPEN Gripper
        PulseDO DO_OPEN_GR;
        WaitTime wait_gripper;

        MoveJ Offs(Target_Base_l2_h2,0,0,0),v1000,fine,Gripper_Fingers;
        !Close gripper
        PulseDO DO_CLOSE_GR;
        WaitTime wait_gripper;

        MoveJ Offs(Target_Base_l2_h2,0,0,100),v1000,fine,Gripper_Fingers;
        MoveJ Offs(Target_Table1_l2_h2,0,0,100),v1000,fine,Gripper_Fingers;
        MoveJ Offs(Target_Table1_l2_h2,0,0,0),v200,fine,Gripper_Fingers;

        PulseDO DO_PROFILE_LOADED;
    ENDPROC

    PROC Big_blocks_backup()
        !OPEN Gripper
        PulseDO DO_OPEN_GR;
        WaitTime wait_gripper;

        MoveJ Offs(Target_Table1_l2_h2,0,0,100),v200,fine,Gripper_Fingers;
        MoveAbsJ Target_JHome,v1000,fine,Gripper_Fingers\WObj:=wobj0;

        PulseDO DO_BACKUPED;
    ENDPROC

    PROC Big_blocks_transfer()
        !OPEN Gripper
        PulseDO DO_OPEN_GR;
        WaitTime wait_gripper;

        MoveJ Offs(Target_Table1_l2_h2,0,0,100),v1000,fine,Gripper_Fingers;
        MoveJ Target_Table1_l2_h2,v200,fine,Gripper_Fingers;
        WaitTime 0.5;

        PulseDO DO_OPEN_TAB1_L;
        PulseDO DO_OPEN_TAB1_R;

        !Close gripper
        PulseDO DO_CLOSE_GR;
        WaitTime wait_gripper;

        MoveL Target_Table1_l2_h2_takeout,v200,fine,Gripper_Fingers;
        MoveL Offs(Target_Table1_l2_h2_takeout,0,0,100),v1000,fine,Gripper_Fingers;

        MoveL Offs(Target_Table2_l2_h2_takeout,0,0,100),v1000,fine,Gripper_Fingers;
        MoveL Offs(Target_Table2_l2_h2_takeout,0,0,0),v200,fine,Gripper_Fingers;
        MoveL Offs(Target_Table2_l2_h2,0,0,0),v200,fine,Gripper_Fingers;

        !Detach
        PulseDO DO_CLOSE_TAB2_L;
        PulseDO DO_CLOSE_TAB2_R;

        PulseDO DO_OPEN_GR;
        WaitTime wait_gripper;

        MoveL Offs(Target_Table2_l2_h2,0,0,100),v1000,fine,Gripper_Fingers;
        MoveAbsJ Target_JHome,v1000,fine,Gripper_Fingers\WObj:=wobj0;

        PulseDO DO_TRANSFERED;
    ENDPROC
    PROC Sync()
        MoveAbsJ Target_JHome,v1000,fine,Gripper_Fingers\WObj:=wobj0;
        MoveL Target_Base_l1_h1,v1000,z100,Gripper_Fingers\WObj:=wobj0;
        MoveL Target_Base_l2_h2,v1000,z100,Gripper_Fingers\WObj:=wobj0;
        MoveL Target_Table1_l2_h2,v1000,z100,Gripper_Fingers\WObj:=wobj0;
        MoveL Target_Table2_l1_h1,v1000,z100,Gripper_Fingers\WObj:=wobj0;
        MoveL Target_Table1_l1_h1,v1000,z100,Gripper_Fingers\WObj:=wobj0;
        MoveL Target_Table2_l2_h2,v1000,z100,Gripper_Fingers\WObj:=wobj0;
        MoveL Target_Table2_l2_h2_takeout,v1000,z100,Gripper_Fingers\WObj:=wobj0;
        MoveL Target_Table1_l2_h2_takeout,v1000,z100,Gripper_Fingers\WObj:=wobj0;
        MoveL Target_Table1_l1_h1_takeout,v1000,z100,Gripper_Fingers\WObj:=wobj0;
        MoveL Target_Table2_l1_h1_takeout,v1000,z100,Gripper_Fingers\WObj:=wobj0;
    ENDPROC
ENDMODULE

--- Controller Data/Controller3/RAPID/TASK1/PROGMOD/CalibData.mod ---
MODULE CalibData
    PERS tooldata Weldgun:=[TRUE,[[20.31,0,363.689],[0.948464781,0,0.316882565,0]],[1,[0,0,1],[1,0,0,0],0,0,0]];
ENDMODULE

--- Controller Data/Controller3/RAPID/TASK1/PROGMOD/Module1.mod ---
MODULE Module1
    CONST jointtarget Target_Idle:=[[0,-70,60,0,45,0],[9E+09,9E+09,9E+09,9E+09,9E+09,9E+09]];

    CONST robtarget Target_20_2:=[[711.495384789,-192.569070764,340],[0.270598049,0.653281483,-0.653281483,0.27059805],[-1,-1,-2,0],[9E+09,9E+09,9E+09,9E+09,9E+09,9E+09]];
    CONST robtarget Target_30_2:=[[756.495384789,-192.569070764,340],[0.270598049,0.653281483,-0.653281483,0.27059805],[-1,-1,-2,0],[9E+09,9E+09,9E+09,9E+09,9E+09,9E+09]];
    CONST robtarget Target_30:=[[756.495384789,-192.569070764,340],[0.45999152,0.077308088,-0.883635489,0.040244043],[-1,-1,-1,0],[9E+09,9E+09,9E+09,9E+09,9E+09,9E+09]];
    CONST robtarget Target_40:=[[756.495384789,-237.569070764,340],[0.382683432,0,-0.923879533,0],[-1,-1,-1,0],[9E+09,9E+09,9E+09,9E+09,9E+09,9E+09]];
    CONST robtarget Target_40_2:=[[756.495384789,-237.569070764,340],[0.27059805,-0.653281483,-0.653281483,-0.27059805],[-1,0,0,0],[9E+09,9E+09,9E+09,9E+09,9E+09,9E+09]];
    CONST robtarget Target_10_2:=[[711.495384789,-237.569070764,340],[0.270598048,-0.653281483,-0.653281483,-0.27059805],[-1,0,0,0],[9E+09,9E+09,9E+09,9E+09,9E+09,9E+09]];
    CONST robtarget Target_10:=[[711.495384789,-237.569070764,340],[0.176703546,-0.819491154,-0.33944435,-0.426600093],[-1,0,1,0],[9E+09,9E+09,9E+09,9E+09,9E+09,9E+09]];
    CONST robtarget Target_20:=[[711.495384789,-192.569070764,340],[-0.000000001,0.923879533,0,0.382683432],[-1,0,1,0],[9E+09,9E+09,9E+09,9E+09,9E+09,9E+09]];
    CONST robtarget Target_10_30_0:=[[614.316010633,-38.379402252,476.187474664],[0.146446608,-0.853553391,-0.353553391,-0.353553391],[-1,0,1,0],[9E+09,9E+09,9E+09,9E+09,9E+09,9E+09]];
    CONST robtarget Target_10_30_1:=[[731.697116217,-72.603148817,474.139403279],[0.379409522,-0.049950211,-0.915975615,0.120590478],[-1,-1,-1,0],[9E+09,9E+09,9E+09,9E+09,9E+09,9E+09]];

    VAR speeddata welding := v150;
    CONST num PType1Offs:=0;
    CONST num PType2Offs:=5;

    VAR bool ColdStart:=TRUE;
    VAR num PTypeRequested;

    PROC main()
        IF ColdStart THEN
            SetDO DO_Weld_IsReady,0;
            SetDO DO_Weld_IsBusy,1;

            MoveAbsJ Target_Idle,v1000,fine,Weldgun\WObj:=wobj0;

            SetDO DO_Weld_IsReady,1;
            SetDO DO_Weld_IsBusy,0;
            ColdStart := FALSE;
        ENDIF

        WaitDI DI_Weld_Stage1Req,1;

        IF TestDI(DI_Weld_ProgT1) THEN
            PTypeRequested:=1;
        ELSEIF TestDI(DI_Weld_ProgT2) THEN
            PTypeRequested:=2;
        ENDIF

        SetDO DO_Weld_IsReady,0;
        SetDO DO_Weld_IsBusy,1;

        PulseDO DO_Weld_1StageEnter;
        Path_10_30 PTypeRequested;
        PulseDO DO_Weld_1StageLeave;

        WaitDI DI_Weld_Stage2Req,1;

        PulseDO DO_Weld_2StageEnter;
        Path_20_30_40_10 PTypeRequested;
        PulseDO DO_Weld_2StageLeave;

        SetDO DO_Weld_IsBusy,0;
        SetDO DO_Weld_IsReady,1;
    ENDPROC

    FUNC robtarget ResolvePtype(robtarget Target,num PType)
        TEST PType
        CASE 1:
            RETURN Offs(Target,0,PType1Offs,0);
        CASE 2:
            RETURN Offs(Target,0,PType2Offs,0);
        DEFAULT:
            RETURN Target;
        ENDTEST
    ENDFUNC

    PROC Path_20_30_40_10(num PType)
        MoveAbsJ Target_Idle,v1000,fine,Weldgun\WObj:=wobj0;

        MoveL Target_10_30_1,v1000,z50,Weldgun\WObj:=wobj0;
        MoveL Offs(Target_20_2,0,10,10),v1000,z100,Weldgun\WObj:=wobj0;

        WaitTime 1;
        MoveL ResolvePtype(Target_20_2,PType),welding,z100,Weldgun\WObj:=wobj0;
        MoveL ResolvePtype(Target_30_2,PType),welding,z100,Weldgun\WObj:=wobj0;
        WaitTime 1;

        MoveL ResolvePtype(Target_30,PType),welding,z100,Weldgun\WObj:=wobj0;
        MoveL ResolvePtype(Target_40,PType),welding,z100,Weldgun\WObj:=wobj0;
        WaitTime 1;
        MoveL ResolvePtype(Target_40_2,PType),welding,z100,Weldgun\WObj:=wobj0;
        MoveL ResolvePtype(Target_10_2,PType),welding,z100,Weldgun\WObj:=wobj0;
        WaitTime 1;
        MoveL ResolvePtype(Target_10,PType),welding,z100,Weldgun\WObj:=wobj0;
        MoveL ResolvePtype(Target_20,PType),welding,z100,Weldgun\WObj:=wobj0;

        MoveL Target_10_30_0,v1000,z50,Weldgun\WObj:=wobj0;

        MoveAbsJ Target_Idle,v1000,fine,Weldgun\WObj:=wobj0;
    ENDPROC

    PROC Path_10_30(num PType)
        MoveAbsJ Target_Idle,v1000,fine,Weldgun\WObj:=wobj0;

        MoveL Target_10_30_0,v1000,z10,Weldgun\WObj:=wobj0;

        MoveL ResolvePtype(Offs(Target_10,-10,0,10),PType),v800,fine,Weldgun\WObj:=wobj0;
        MoveL ResolvePtype(Target_10,PType),welding,fine,Weldgun\WObj:=wobj0;
        WaitTime 0.5;
        MoveL ResolvePtype(Offs(Target_10,-10,0,10),PType),welding,fine,Weldgun\WObj:=wobj0;

        MoveL Target_10_30_0,v1000,z10,Weldgun\WObj:=wobj0;
        MoveL Target_10_30_1,v1000,z10,Weldgun\WObj:=wobj0;

        MoveL ResolvePtype(Offs(Target_30,10,10,10),PType),v800,fine,Weldgun\WObj:=wobj0;
        MoveL ResolvePtype(Target_30,PType),welding,fine,Weldgun\WObj:=wobj0;
        WaitTime 0.5;
        MoveL ResolvePtype(Offs(Target_30,10,10,10),PType),welding,fine,Weldgun\WObj:=wobj0;

        MoveL Target_10_30_1,v1000,z10,Weldgun\WObj:=wobj0;
        MoveAbsJ Target_Idle,v1000,fine,Weldgun\WObj:=wobj0;
    ENDPROC

    PROC Path_10_20()
        MoveL Target_10,welding,fine,Weldgun\WObj:=wobj0;
        MoveL Target_20,welding,fine,Weldgun\WObj:=wobj0;
    ENDPROC

    PROC Path_20_30()
        MoveL Target_20_2,welding,fine,Weldgun\WObj:=wobj0;
        MoveL Target_30_2,welding,fine,Weldgun\WObj:=wobj0;
    ENDPROC

    PROC Path_30_40()
        MoveL Target_30,welding,fine,Weldgun\WObj:=wobj0;
        MoveL Target_40,welding,fine,Weldgun\WObj:=wobj0;
    ENDPROC

    PROC Path_40_10()
        MoveL Target_10_2,welding,fine,Weldgun\WObj:=wobj0;
        MoveL Target_40_2,welding,fine,Weldgun\WObj:=wobj0;
    ENDPROC
    PROC Sync()
        MoveL Target_10,v1000,z100,Weldgun\WObj:=wobj0;
        MoveL Target_10_2,v1000,z100,Weldgun\WObj:=wobj0;
        MoveL Target_10_30_0,v1000,z100,Weldgun\WObj:=wobj0;
        MoveL Target_10_30_1,v1000,z100,Weldgun\WObj:=wobj0;
        MoveL Target_20,v1000,z100,Weldgun\WObj:=wobj0;
        MoveL Target_20_2,v1000,z100,Weldgun\WObj:=wobj0;
        MoveL Target_30,v1000,z100,Weldgun\WObj:=wobj0;
        MoveL Target_30_2,v1000,z100,Weldgun\WObj:=wobj0;
        MoveL Target_40,v1000,z100,Weldgun\WObj:=wobj0;
        MoveL Target_40_2,v1000,z100,Weldgun\WObj:=wobj0;
    ENDPROC
ENDMODULE

--- Controller Data/Controller4/RAPID/TASK1/PROGMOD/CalibData.mod ---
MODULE CalibData
    PERS tooldata Drill_Tool:=[TRUE,[[211.187000005,0.000000004,132.999999995],[0.707106781,0,0.707106781,0]],[1,[-40.884000001,0.010000002,112.464],[1,0,0,0],0,0,0]];
ENDMODULE

--- Controller Data/Controller4/RAPID/TASK1/PROGMOD/Module1.mod ---
MODULE Module1
    CONST robtarget T_Drill_aHome:=[[457.561710524,-9.948272227,1001.147802577],[0.173648178,0,-0.984807753,0],[0,0,0,0],[9E+09,9E+09,9E+09,9E+09,9E+09,9E+09]];
    CONST robtarget T_Drill_COM_10:=[[905.457950428,-195,345.666062685],[0.160429997,-0.376869611,-0.909843726,0.066452281],[0,-1,1,0],[9E+09,9E+09,9E+09,9E+09,9E+09,9E+09]];
    CONST robtarget T_Drill_COM_20:=[[943.045950428,-195,331.985062685],[0.160429997,-0.376869611,-0.909843726,0.066452281],[0,-1,1,0],[9E+09,9E+09,9E+09,9E+09,9E+09,9E+09]];
    CONST robtarget T_Drill_S_30:=[[943.045950428,-125,331.985062685],[0.160429997,-0.376869611,-0.909843726,0.066452281],[0,-1,1,0],[9E+09,9E+09,9E+09,9E+09,9E+09,9E+09]];
    CONST robtarget T_Drill_S_40:=[[905.457950428,-125,345.666062685],[0.160429997,-0.376869611,-0.909843726,0.066452281],[0,-1,1,0],[9E+09,9E+09,9E+09,9E+09,9E+09,9E+09]];
    CONST robtarget T_Drill_L_30:=[[943.045950428,-115,331.985062685],[0.160429997,-0.376869611,-0.909843726,0.066452281],[0,-1,1,0],[9E+09,9E+09,9E+09,9E+09,9E+09,9E+09]];
    CONST robtarget T_Drill_L_40:=[[905.457950428,-115,345.666062685],[0.160429997,-0.376869611,-0.909843726,0.066452281],[0,-1,1,0],[9E+09,9E+09,9E+09,9E+09,9E+09,9E+09]];

    VAR speeddata vel_move := v800;
    VAR speeddata vel_drill := v50;
    VAR speeddata vel_gotohole := v500;
    VAR num offset := -250;
    VAR num drillhole := 7;

    VAR bool COLD_START:=TRUE;

    PROC main()
        IF COLD_START THEN
            MoveL RelTool(T_Drill_aHome, 0, 0, 0),vel_move,fine,Drill_Tool\WObj:=wobj0;
            COLD_START := FALSE;
            SetDO DO_DRILL_READY,1;
        ENDIF

        WaitDI DI_EXEC_DRILL,1;
        SetDO DO_DRILL_READY,0;

        IF TestDI(DI_PTYPE_1) THEN
            Path_Drill_S;
            MoveL RelTool(T_Drill_aHome, 0, 0, 0),vel_move,fine,Drill_Tool\WObj:=wobj0;
            PulseDO DO_DRILL_DONE;
        ELSEIF TestDI(DI_PTYPE_2) THEN
            Path_Drill_L;
            MoveL RelTool(T_Drill_aHome, 0, 0, 0),vel_move,fine,Drill_Tool\WObj:=wobj0;
            PulseDO DO_DRILL_DONE;
        ELSE
            RETURN ;
        ENDIF
    ENDPROC

    PROC Path_Drill_S()
        MoveL RelTool(T_Drill_COM_10, 0, 0, offset),vel_move,fine,Drill_Tool\WObj:=wobj0;
        MoveL RelTool(T_Drill_COM_10, 0, 0, 0),vel_gotohole,fine,Drill_Tool\WObj:=wobj0;
        WaitTime 0.5;
        MoveL RelTool(T_Drill_COM_10, 0, 0, drillhole),vel_drill,fine,Drill_Tool\WObj:=wobj0;
        MoveL RelTool(T_Drill_COM_10, 0, 0, 0),vel_drill,fine,Drill_Tool\WObj:=wobj0;
        WaitTime 0.5;
        MoveL RelTool(T_Drill_COM_10, 0, 0, offset),vel_gotohole,fine,Drill_Tool\WObj:=wobj0;

        MoveL RelTool(T_Drill_COM_20, 0, 0, offset),vel_move,fine,Drill_Tool\WObj:=wobj0;
        MoveL RelTool(T_Drill_COM_20, 0, 0, 0),vel_gotohole,fine,Drill_Tool\WObj:=wobj0;
        WaitTime 0.5;
        MoveL RelTool(T_Drill_COM_20, 0, 0, drillhole),vel_drill,fine,Drill_Tool\WObj:=wobj0;
        MoveL RelTool(T_Drill_COM_20, 0, 0, 0),vel_drill,fine,Drill_Tool\WObj:=wobj0;
        WaitTime 0.5;
        MoveL RelTool(T_Drill_COM_20, 0, 0, offset),vel_gotohole,fine,Drill_Tool\WObj:=wobj0;

        MoveL RelTool(T_Drill_S_30, 0, 0, offset),vel_move,fine,Drill_Tool\WObj:=wobj0;
        MoveL RelTool(T_Drill_S_30, 0, 0, 0),vel_gotohole,fine,Drill_Tool\WObj:=wobj0;
        WaitTime 0.5;
        MoveL RelTool(T_Drill_S_30, 0, 0, drillhole),vel_drill,fine,Drill_Tool\WObj:=wobj0;
        MoveL RelTool(T_Drill_S_30, 0, 0, 0),vel_drill,fine,Drill_Tool\WObj:=wobj0;
        WaitTime 0.5;
        MoveL RelTool(T_Drill_S_30, 0, 0, offset),vel_gotohole,fine,Drill_Tool\WObj:=wobj0;

        MoveL RelTool(T_Drill_S_40, 0, 0, offset),vel_move,fine,Drill_Tool\WObj:=wobj0;
        MoveL RelTool(T_Drill_S_40, 0, 0, 0),vel_gotohole,fine,Drill_Tool\WObj:=wobj0;
        WaitTime 0.5;
        MoveL RelTool(T_Drill_S_40, 0, 0, drillhole),vel_drill,fine,Drill_Tool\WObj:=wobj0;
        MoveL RelTool(T_Drill_S_40, 0, 0, 0),vel_drill,fine,Drill_Tool\WObj:=wobj0;
        WaitTime 0.5;
        MoveL RelTool(T_Drill_S_40, 0, 0, offset),vel_gotohole,fine,Drill_Tool\WObj:=wobj0;

        !MoveL T_Drill_aHome,v200,fine,Drill_Tool\WObj:=wobj0;
        !MoveL T_Drill_COM_10,v200,fine,Drill_Tool\WObj:=wobj0;
        !MoveL T_Drill_COM_20,v200,fine,Drill_Tool\WObj:=wobj0;
        !MoveL T_Drill_S_30,v200,fine,Drill_Tool\WObj:=wobj0;
        !MoveL T_Drill_S_40,v200,fine,Drill_Tool\WObj:=wobj0;
    ENDPROC

    PROC Path_Drill_L()
        MoveL RelTool(T_Drill_COM_10, 0, 0, offset),vel_move,fine,Drill_Tool\WObj:=wobj0;
        MoveL RelTool(T_Drill_COM_10, 0, 0, 0),vel_gotohole,fine,Drill_Tool\WObj:=wobj0;
        WaitTime 0.5;
        MoveL RelTool(T_Drill_COM_10, 0, 0, drillhole),vel_drill,fine,Drill_Tool\WObj:=wobj0;
        MoveL RelTool(T_Drill_COM_10, 0, 0, 0),vel_drill,fine,Drill_Tool\WObj:=wobj0;
        WaitTime 0.5;
        MoveL RelTool(T_Drill_COM_10, 0, 0, offset),vel_gotohole,fine,Drill_Tool\WObj:=wobj0;

        MoveL RelTool(T_Drill_COM_20, 0, 0, offset),vel_move,fine,Drill_Tool\WObj:=wobj0;
        MoveL RelTool(T_Drill_COM_20, 0, 0, 0),vel_gotohole,fine,Drill_Tool\WObj:=wobj0;
        WaitTime 0.5;
        MoveL RelTool(T_Drill_COM_20, 0, 0, drillhole),vel_drill,fine,Drill_Tool\WObj:=wobj0;
        MoveL RelTool(T_Drill_COM_20, 0, 0, 0),vel_drill,fine,Drill_Tool\WObj:=wobj0;
        WaitTime 0.5;
        MoveL RelTool(T_Drill_COM_20, 0, 0, offset),vel_gotohole,fine,Drill_Tool\WObj:=wobj0;

        MoveL RelTool(T_Drill_L_30, 0, 0, offset),vel_move,fine,Drill_Tool\WObj:=wobj0;
        MoveL RelTool(T_Drill_L_30, 0, 0, 0),vel_gotohole,fine,Drill_Tool\WObj:=wobj0;
        WaitTime 0.5;
        MoveL RelTool(T_Drill_L_30, 0, 0, drillhole),vel_drill,fine,Drill_Tool\WObj:=wobj0;
        MoveL RelTool(T_Drill_L_30, 0, 0, 0),vel_drill,fine,Drill_Tool\WObj:=wobj0;
        WaitTime 0.5;
        MoveL RelTool(T_Drill_L_30, 0, 0, offset),vel_gotohole,fine,Drill_Tool\WObj:=wobj0;

        MoveL RelTool(T_Drill_L_40, 0, 0, offset),vel_move,fine,Drill_Tool\WObj:=wobj0;
        MoveL RelTool(T_Drill_L_40, 0, 0, 0),vel_gotohole,fine,Drill_Tool\WObj:=wobj0;
        WaitTime 0.5;
        MoveL RelTool(T_Drill_L_40, 0, 0, drillhole),vel_drill,fine,Drill_Tool\WObj:=wobj0;
        MoveL RelTool(T_Drill_L_40, 0, 0, 0),vel_drill,fine,Drill_Tool\WObj:=wobj0;
        WaitTime 0.5;
        MoveL RelTool(T_Drill_L_40, 0, 0, offset),vel_gotohole,fine,Drill_Tool\WObj:=wobj0;

        !MoveL T_Drill_aHome,v200,fine,Drill_Tool\WObj:=wobj0;
        !MoveL T_Drill_COM_10,v200,fine,Drill_Tool\WObj:=wobj0;
        !MoveL T_Drill_COM_20,v200,fine,Drill_Tool\WObj:=wobj0;
        !MoveL T_Drill_L_30,v200,fine,Drill_Tool\WObj:=wobj0;
        !MoveL T_Drill_L_40,v200,fine,Drill_Tool\WObj:=wobj0;
    ENDPROC

    PROC Sync()
        MoveL T_Drill_aHome,v200,fine,Drill_Tool\WObj:=wobj0;
        MoveL T_Drill_COM_10,v200,fine,Drill_Tool\WObj:=wobj0;
        MoveL T_Drill_COM_20,v200,fine,Drill_Tool\WObj:=wobj0;
        MoveL T_Drill_S_30,v200,fine,Drill_Tool\WObj:=wobj0;
        MoveL T_Drill_S_40,v200,fine,Drill_Tool\WObj:=wobj0;
        MoveL T_Drill_L_30,v200,fine,Drill_Tool\WObj:=wobj0;
        MoveL T_Drill_L_40,v200,fine,Drill_Tool\WObj:=wobj0;
    ENDPROC

ENDMODULE

--- Controller Data/Controller4/RAPID/TASK2/PROGMOD/CalibData.mod ---
MODULE CalibData
    PERS tooldata Endeep_Tool:=[TRUE,[[257.929,0,133],[0.707106781,0,0.707106781,0]],[1,[40.263,-0.01,112.48],[1,0,0,0],0,0,0]];
ENDMODULE

--- Controller Data/Controller4/RAPID/TASK2/PROGMOD/Module1.mod ---
MODULE Module1
    CONST robtarget T_Endeep_aHome:=[[797.552204235,-362.673625766,1349.391204212],[0,0.984807753,0,-0.173648178],[0,0,0,0],[9E+09,9E+09,9E+09,9E+09,9E+09,9E+09]];
    CONST robtarget T_Endeep_COM_10:=[[905.458,-195,345.666],[0,0.984807753,0,-0.173648178],[-1,0,-2,0],[9E+09,9E+09,9E+09,9E+09,9E+09,9E+09]];
    CONST robtarget T_Endeep_COM_20:=[[943.046,-195,331.985],[0,0.984807753,0,-0.173648178],[-1,0,-2,0],[9E+09,9E+09,9E+09,9E+09,9E+09,9E+09]];
    CONST robtarget T_Endeep_S_30:=[[943.046,-125,331.985],[0,0.984807753,0,-0.173648178],[-1,0,-2,0],[9E+09,9E+09,9E+09,9E+09,9E+09,9E+09]];
    CONST robtarget T_Endeep_S_40:=[[905.458,-125,345.666],[0,0.984807753,0,-0.173648178],[-1,0,-2,0],[9E+09,9E+09,9E+09,9E+09,9E+09,9E+09]];
    CONST robtarget T_Endeep_L_30:=[[943.046,-115,331.985],[0,0.984807753,0,-0.173648178],[-1,0,-2,0],[9E+09,9E+09,9E+09,9E+09,9E+09,9E+09]];
    CONST robtarget T_Endeep_L_40:=[[905.458,-115,345.666],[0,0.984807753,0,-0.173648178],[-1,0,-2,0],[9E+09,9E+09,9E+09,9E+09,9E+09,9E+09]];

    VAR speeddata vel_move:=v800;
    VAR speeddata vel_drill:=v50;
    VAR speeddata vel_gotohole:=v500;
    VAR num offset:=-250;
    VAR num endeephole:=2.5;

    VAR bool COLD_START:=TRUE;

    PROC main()
        IF COLD_START THEN
            MoveL RelTool(T_Endeep_aHome, 0, 0, 0),vel_move,fine,Endeep_Tool\WObj:=wobj0;
            COLD_START := FALSE;
        ENDIF

        WaitDI DI_EXEC_ENDEEP,1;

        IF TestDI(DI_PTYPE_1) THEN
            Path_Endeep_S;
            MoveL RelTool(T_Endeep_aHome, 0, 0, 0),vel_move,fine,Endeep_Tool\WObj:=wobj0;
            PulseDO DO_ENDEEP_DONE;
        ELSEIF TestDI(DI_PTYPE_2) THEN
            Path_Endeep_L;
            MoveL RelTool(T_Endeep_aHome, 0, 0, 0),vel_move,fine,Endeep_Tool\WObj:=wobj0;
            PulseDO DO_ENDEEP_DONE;
        ELSE
            RETURN ;
        ENDIF

        PulseDO DO_ENDEEP_DONE;
        SetDO DO_DRILL_READY,1;

    ENDPROC

    PROC Path_Endeep_S()
        MoveL RelTool(T_Endeep_COM_10,0,0,offset),vel_move,fine,Endeep_Tool\WObj:=wobj0;
        MoveL RelTool(T_Endeep_COM_10,0,0,0),vel_gotohole,fine,Endeep_Tool\WObj:=wobj0;
        WaitTime 0.5;
        MoveL RelTool(T_Endeep_COM_10,0,0,endeephole),vel_drill,fine,Endeep_Tool\WObj:=wobj0;
        MoveL RelTool(T_Endeep_COM_10,0,0,0),vel_drill,fine,Endeep_Tool\WObj:=wobj0;
        WaitTime 0.5;
        MoveL RelTool(T_Endeep_COM_10,0,0,offset),vel_gotohole,fine,Endeep_Tool\WObj:=wobj0;

        MoveL RelTool(T_Endeep_COM_20,0,0,offset),vel_move,fine,Endeep_Tool\WObj:=wobj0;
        MoveL RelTool(T_Endeep_COM_20,0,0,0),vel_gotohole,fine,Endeep_Tool\WObj:=wobj0;
        WaitTime 0.5;
        MoveL RelTool(T_Endeep_COM_20,0,0,endeephole),vel_drill,fine,Endeep_Tool\WObj:=wobj0;
        MoveL RelTool(T_Endeep_COM_20,0,0,0),vel_drill,fine,Endeep_Tool\WObj:=wobj0;
        WaitTime 0.5;
        MoveL RelTool(T_Endeep_COM_20,0,0,offset),vel_gotohole,fine,Endeep_Tool\WObj:=wobj0;

        MoveL RelTool(T_Endeep_S_30,0,0,offset),vel_move,fine,Endeep_Tool\WObj:=wobj0;
        MoveL RelTool(T_Endeep_S_30,0,0,0),vel_gotohole,fine,Endeep_Tool\WObj:=wobj0;
        WaitTime 0.5;
        MoveL RelTool(T_Endeep_S_30,0,0,endeephole),vel_drill,fine,Endeep_Tool\WObj:=wobj0;
        MoveL RelTool(T_Endeep_S_30,0,0,0),vel_drill,fine,Endeep_Tool\WObj:=wobj0;
        WaitTime 0.5;
        MoveL RelTool(T_Endeep_S_30,0,0,offset),vel_gotohole,fine,Endeep_Tool\WObj:=wobj0;

        MoveL RelTool(T_Endeep_S_40,0,0,offset),vel_move,fine,Endeep_Tool\WObj:=wobj0;
        MoveL RelTool(T_Endeep_S_40,0,0,0),vel_gotohole,fine,Endeep_Tool\WObj:=wobj0;
        WaitTime 0.5;
        MoveL RelTool(T_Endeep_S_40,0,0,endeephole),vel_drill,fine,Endeep_Tool\WObj:=wobj0;
        MoveL RelTool(T_Endeep_S_40,0,0,0),vel_drill,fine,Endeep_Tool\WObj:=wobj0;
        WaitTime 0.5;
        MoveL RelTool(T_Endeep_S_40,0,0,offset),vel_gotohole,fine,Endeep_Tool\WObj:=wobj0;

        !MoveL T_Endeep_aHome,v200,fine,Endeep_Tool\WObj:=wobj0;
        !MoveL T_Endeep_COM_10,v200,fine,Endeep_Tool\WObj:=wobj0;
        !MoveL T_Endeep_COM_20,v200,fine,Endeep_Tool\WObj:=wobj0;
        !MoveL T_Endeep_S_30,v200,fine,Endeep_Tool\WObj:=wobj0;
        !MoveL T_Endeep_S_40,v200,fine,Endeep_Tool\WObj:=wobj0;
    ENDPROC

    PROC Path_Endeep_L()
        MoveL RelTool(T_Endeep_COM_10,0,0,offset),vel_move,fine,Endeep_Tool\WObj:=wobj0;
        MoveL RelTool(T_Endeep_COM_10,0,0,0),vel_gotohole,fine,Endeep_Tool\WObj:=wobj0;
        WaitTime 0.5;
        MoveL RelTool(T_Endeep_COM_10,0,0,endeephole),vel_drill,fine,Endeep_Tool\WObj:=wobj0;
        MoveL RelTool(T_Endeep_COM_10,0,0,0),vel_drill,fine,Endeep_Tool\WObj:=wobj0;
        WaitTime 0.5;
        MoveL RelTool(T_Endeep_COM_10,0,0,offset),vel_gotohole,fine,Endeep_Tool\WObj:=wobj0;

        MoveL RelTool(T_Endeep_COM_20,0,0,offset),vel_move,fine,Endeep_Tool\WObj:=wobj0;
        MoveL RelTool(T_Endeep_COM_20,0,0,0),vel_gotohole,fine,Endeep_Tool\WObj:=wobj0;
        WaitTime 0.5;
        MoveL RelTool(T_Endeep_COM_20,0,0,endeephole),vel_drill,fine,Endeep_Tool\WObj:=wobj0;
        MoveL RelTool(T_Endeep_COM_20,0,0,0),vel_drill,fine,Endeep_Tool\WObj:=wobj0;
        WaitTime 0.5;
        MoveL RelTool(T_Endeep_COM_20,0,0,offset),vel_gotohole,fine,Endeep_Tool\WObj:=wobj0;

        MoveL RelTool(T_Endeep_L_30,0,0,offset),vel_move,fine,Endeep_Tool\WObj:=wobj0;
        MoveL RelTool(T_Endeep_L_30,0,0,0),vel_gotohole,fine,Endeep_Tool\WObj:=wobj0;
        WaitTime 0.5;
        MoveL RelTool(T_Endeep_L_30,0,0,endeephole),vel_drill,fine,Endeep_Tool\WObj:=wobj0;
        MoveL RelTool(T_Endeep_L_30,0,0,0),vel_drill,fine,Endeep_Tool\WObj:=wobj0;
        WaitTime 0.5;
        MoveL RelTool(T_Endeep_L_30,0,0,offset),vel_gotohole,fine,Endeep_Tool\WObj:=wobj0;

        MoveL RelTool(T_Endeep_L_40,0,0,offset),vel_move,fine,Endeep_Tool\WObj:=wobj0;
        MoveL RelTool(T_Endeep_L_40,0,0,0),vel_gotohole,fine,Endeep_Tool\WObj:=wobj0;
        WaitTime 0.5;
        MoveL RelTool(T_Endeep_L_40,0,0,endeephole),vel_drill,fine,Endeep_Tool\WObj:=wobj0;
        MoveL RelTool(T_Endeep_L_40,0,0,0),vel_drill,fine,Endeep_Tool\WObj:=wobj0;
        WaitTime 0.5;
        MoveL RelTool(T_Endeep_L_40,0,0,offset),vel_gotohole,fine,Endeep_Tool\WObj:=wobj0;

        !MoveL T_Endeep_aHome,v200,fine,Endeep_Tool\WObj:=wobj0;
        !MoveL T_Endeep_COM_10,v200,fine,Endeep_Tool\WObj:=wobj0;
        !MoveL T_Endeep_COM_20,v200,fine,Endeep_Tool\WObj:=wobj0;
        !MoveL T_Endeep_L_30,v200,fine,Endeep_Tool\WObj:=wobj0;
        !MoveL T_Endeep_L_40,v200,fine,Endeep_Tool\WObj:=wobj0;
    ENDPROC

    PROC Sync()
        MoveL T_Endeep_aHome,v200,fine,Endeep_Tool\WObj:=wobj0;
        MoveL T_Endeep_COM_10,v200,fine,Endeep_Tool\WObj:=wobj0;
        MoveL T_Endeep_COM_20,v200,fine,Endeep_Tool\WObj:=wobj0;
        MoveL T_Endeep_S_30,v200,fine,Endeep_Tool\WObj:=wobj0;
        MoveL T_Endeep_S_40,v200,fine,Endeep_Tool\WObj:=wobj0;
        MoveL T_Endeep_L_30,v200,fine,Endeep_Tool\WObj:=wobj0;
        MoveL T_Endeep_L_40,v200,fine,Endeep_Tool\WObj:=wobj0;
    ENDPROC
ENDMODULE

--- Controller Data/Controller1/SYSPAR/EIO.cfg ---
EIO:CFG_1.0:6:1::
#
EIO_SIGNAL:

      -Name "DO_OPEN_TAB1_L" -SignalType "DO"

      -Name "DO_OPEN_TAB1_R" -SignalType "DO"

      -Name "DO_CLOSE_TAB1_L" -SignalType "DO"

      -Name "DO_CLOSE_TAB1_R" -SignalType "DO"

      -Name "DO_CLOSE_TAB2_L" -SignalType "DO"

      -Name "DO_CLOSE_TAB2_R" -SignalType "DO"

      -Name "DO_OPEN_TAB2_L" -SignalType "DO"

      -Name "DO_OPEN_TAB2_R" -SignalType "DO"

      -Name "DO_OPEN_GR" -SignalType "DO"

      -Name "DO_CLOSE_GR" -SignalType "DO"

      -Name "DI_PTYPE_2" -SignalType "DI"

      -Name "DI_PTYPE_1" -SignalType "DI"

      -Name "DI_EXEC_LOAD_DESK" -SignalType "DI"

      -Name "DI_EXEC_LOAD_PROFILE" -SignalType "DI"

      -Name "DI_EXEC_TRANSFER" -SignalType "DI"

      -Name "DO_VACUUM_ON" -SignalType "DO"

      -Name "DO_VACUUM_OFF" -SignalType "DO"

      -Name "DO_DESK_LOADED" -SignalType "DO"

      -Name "DO_PROFILE_LOADED" -SignalType "DO"

      -Name "DI_EXEC_BACKUP" -SignalType "DI"

      -Name "DO_BACKUPED" -SignalType "DO"

      -Name "DO_TRANSFERED" -SignalType "DO"

      -Name "DI_ALLOW_LOAD" -SignalType "DI"

      -Name "DI_ALLOW_TRANSFER" -SignalType "DI"

--- Controller Data/Controller3/SYSPAR/EIO.cfg ---
EIO:CFG_1.0:6:1::
#
EIO_SIGNAL:

      -Name "DO_Weld_IsReady" -SignalType "DO"

      -Name "DO_Weld_IsBusy" -SignalType "DO"

      -Name "DO_Weld_1StageWip" -SignalType "DO"

      -Name "DO_Weld_2StageWip" -SignalType "DO"

      -Name "DO_Weld_1StageEnter" -SignalType "DO"

      -Name "DO_Weld_1StageLeave" -SignalType "DO"

      -Name "DO_Weld_2StageEnter" -SignalType "DO"

      -Name "DO_Weld_2StageLeave" -SignalType "DO"

      -Name "DI_Weld_ProgT1" -SignalType "DI"

      -Name "DI_Weld_ProgT2" -SignalType "DI"

      -Name "DI_Weld_Stage2Req" -SignalType "DI"

      -Name "DI_Weld_Stage1Req" -SignalType "DI"

--- Controller Data/Controller4/SYSPAR/EIO.cfg ---
EIO:CFG_1.0:6:1::
#
EIO_SIGNAL:

      -Name "DO_DRILL_DONE" -SignalType "DO"

      -Name "DO_ENDEEP_DONE" -SignalType "DO"

      -Name "DI_EXEC_DRILL" -SignalType "DI"

      -Name "DI_EXEC_ENDEEP" -SignalType "DI"

      -Name "DI_PTYPE_1" -SignalType "DI"

      -Name "DI_PTYPE_2" -SignalType "DI"

      -Name "DO_DRILL_READY" -SignalType "DO"
